SYSTEM CappingStation2
  (* Version 1.0, YYYY-MM-DD, Author, Eclipse 4diac *)
  APPLICATION Application
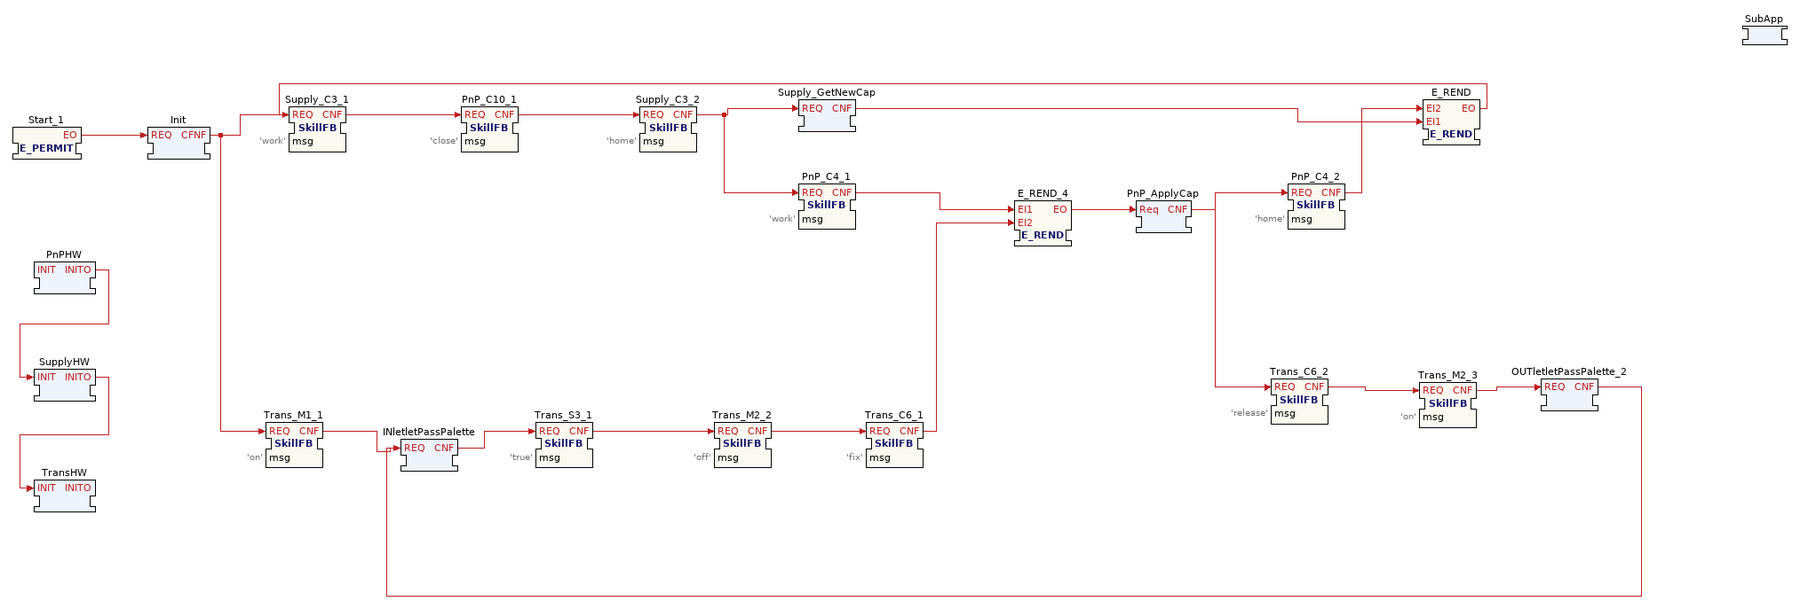
    FBS
      Start_1 : E_PERMIT;
      Supply_C3_1 : SkillFB(msg := 'work');
      Supply_C3_2 : SkillFB(msg := 'home');
      PnP_C10_1 : SkillFB(msg := 'close');
      PnP_C4_1 : SkillFB(msg := 'work');
      Trans_S3_1 : SkillFB(msg := 'true');
      Trans_M1_1 : SkillFB(msg := 'on');
      Trans_M2_2 : SkillFB(msg := 'off');
      Trans_C6_1 : SkillFB(msg := 'fix');
      E_REND_4 : E_REND;
      Trans_C6_2 : SkillFB(msg := 'release');
      Trans_M2_3 : SkillFB(msg := 'on');
      PnP_C4_2 : SkillFB(msg := 'home');
      E_REND : E_REND;
    END_FBS
    SUBAPPLICATION PnPHW
      EVENT_INPUT
        INIT;
      END_EVENT
      EVENT_OUTPUT
        INITO;
      END_EVENT
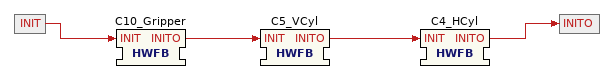
      FBS
        C10_Gripper : HWFB;
        C5_VCyl : HWFB;
        C4_HCyl : HWFB;
      END_FBS
      EVENT_CONNECTIONS
        INIT TO C10_Gripper.INIT;
        C10_Gripper.INITO TO C5_VCyl.INIT;
        C5_VCyl.INITO TO C4_HCyl.INIT;
        C4_HCyl.INITO TO INITO;
      END_CONNECTIONS
    END_SUBAPPLICATION
    SUBAPPLICATION SupplyHW
      EVENT_INPUT
        INIT;
      END_EVENT
      EVENT_OUTPUT
        INITO;
      END_EVENT
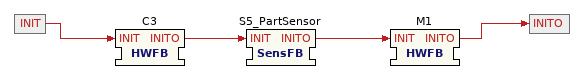
      FBS
        C3 : HWFB;
        M1 : HWFB;
        S5_PartSensor : SensFB;
      END_FBS
      EVENT_CONNECTIONS
        INIT TO C3.INIT;
        M1.INITO TO INITO;
        C3.INITO TO S5_PartSensor.INIT;
        S5_PartSensor.INITO TO M1.INIT;
      END_CONNECTIONS
    END_SUBAPPLICATION
    SUBAPPLICATION TransHW
      EVENT_INPUT
        INIT;
      END_EVENT
      EVENT_OUTPUT
        INITO;
      END_EVENT
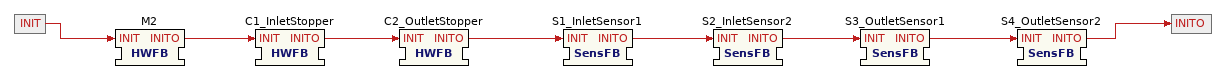
      FBS
        M2 : HWFB;
        C2_OutletStopper : HWFB;
        C1_InletStopper : HWFB;
        S1_InletSensor1 : SensFB;
        S2_InletSensor2 : SensFB;
        S3_OutletSensor1 : SensFB;
        S4_OutletSensor2 : SensFB;
      END_FBS
      EVENT_CONNECTIONS
        INIT TO M2.INIT;
        C1_InletStopper.INITO TO C2_OutletStopper.INIT;
        M2.INITO TO C1_InletStopper.INIT;
        C2_OutletStopper.INITO TO S1_InletSensor1.INIT;
        S1_InletSensor1.INITO TO S2_InletSensor2.INIT;
        S2_InletSensor2.INITO TO S3_OutletSensor1.INIT;
        S3_OutletSensor1.INITO TO S4_OutletSensor2.INIT;
        S4_OutletSensor2.INITO TO INITO;
      END_CONNECTIONS
    END_SUBAPPLICATION
    SUBAPPLICATION SubApp (* All Basic Skills *)
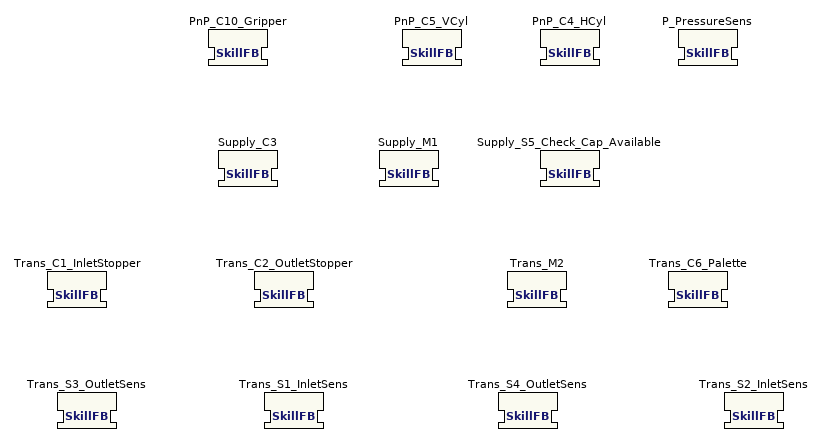
      FBS
        PnP_C10_Gripper : SkillFB;
        PnP_C5_VCyl : SkillFB;
        PnP_C4_HCyl : SkillFB;
        P_PressureSens : SkillFB;
        Supply_C3 : SkillFB;
        Supply_M1 : SkillFB;
        Supply_S5_Check_Cap_Available : SkillFB;
        Trans_C1_InletStopper : SkillFB;
        Trans_C2_OutletStopper : SkillFB;
        Trans_M2 : SkillFB;
        Trans_C6_Palette : SkillFB;
        Trans_S3_OutletSens : SkillFB;
        Trans_S4_OutletSens : SkillFB;
        Trans_S2_InletSens : SkillFB;
        Trans_S1_InletSens : SkillFB;
      END_FBS
    END_SUBAPPLICATION
    SUBAPPLICATION INletletPassPalette (* Composite Skill to let a product pass through the stoper *)
      EVENT_INPUT
        REQ;
      END_EVENT
      EVENT_OUTPUT
        CNF;
      END_EVENT
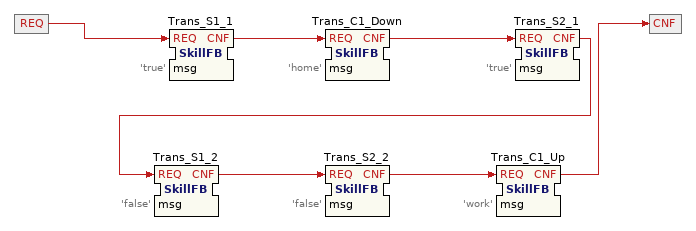
      FBS
        Trans_S1_2 : SkillFB(msg := 'false');
        Trans_S2_2 : SkillFB(msg := 'false');
        Trans_S1_1 : SkillFB(msg := 'true');
        Trans_S2_1 : SkillFB(msg := 'true');
        Trans_C1_Down : SkillFB(msg := 'home');
        Trans_C1_Up : SkillFB(msg := 'work');
      END_FBS
      EVENT_CONNECTIONS
        Trans_S1_2.CNF TO Trans_S2_2.REQ;
        Trans_S1_1.CNF TO Trans_C1_Down.REQ;
        Trans_C1_Down.CNF TO Trans_S2_1.REQ;
        REQ TO Trans_S1_1.REQ;
        Trans_S2_2.CNF TO Trans_C1_Up.REQ;
        Trans_C1_Up.CNF TO CNF;
        Trans_S2_1.CNF TO Trans_S1_2.REQ;
      END_CONNECTIONS
    END_SUBAPPLICATION
    SUBAPPLICATION OUTletletPassPalette_2
      EVENT_INPUT
        REQ;
      END_EVENT
      EVENT_OUTPUT
        CNF;
      END_EVENT
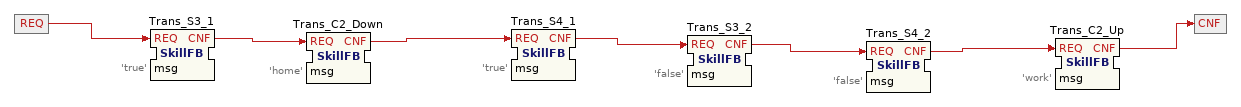
      FBS
        Trans_S3_2 : SkillFB(msg := 'false');
        Trans_S4_2 : SkillFB(msg := 'false');
        Trans_S3_1 : SkillFB(msg := 'true');
        Trans_S4_1 : SkillFB(msg := 'true');
        Trans_C2_Down : SkillFB(msg := 'home');
        Trans_C2_Up : SkillFB(msg := 'work');
      END_FBS
      EVENT_CONNECTIONS
        Trans_S4_1.CNF TO Trans_S3_2.REQ;
        Trans_S3_2.CNF TO Trans_S4_2.REQ;
        Trans_S3_1.CNF TO Trans_C2_Down.REQ;
        Trans_C2_Down.CNF TO Trans_S4_1.REQ;
        REQ TO Trans_S3_1.REQ;
        Trans_S4_2.CNF TO Trans_C2_Up.REQ;
        Trans_C2_Up.CNF TO CNF;
      END_CONNECTIONS
    END_SUBAPPLICATION
    SUBAPPLICATION Init
      EVENT_INPUT
        REQ;
      END_EVENT
      EVENT_OUTPUT
        CFNF;
      END_EVENT
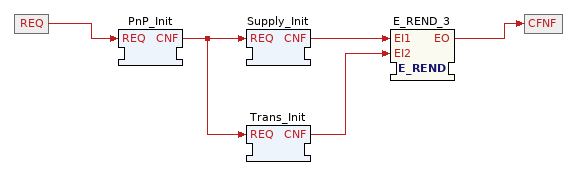
      FBS
        E_REND_3 : E_REND;
      END_FBS
      SUBAPPLICATION Supply_Init
        EVENT_INPUT
          REQ;
        END_EVENT
        EVENT_OUTPUT
          CNF;
        END_EVENT
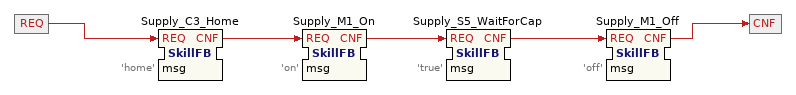
        FBS
          Supply_C3_Home : SkillFB(msg := 'home');
          Supply_M1_Off : SkillFB(msg := 'off');
          Supply_M1_On : SkillFB(msg := 'on');
          Supply_S5_WaitForCap : SkillFB(msg := 'true');
        END_FBS
        EVENT_CONNECTIONS
          Supply_C3_Home.CNF TO Supply_M1_On.REQ;
          Supply_S5_WaitForCap.CNF TO Supply_M1_Off.REQ;
          Supply_M1_On.CNF TO Supply_S5_WaitForCap.REQ;
          REQ TO Supply_C3_Home.REQ;
          Supply_M1_Off.CNF TO CNF;
        END_CONNECTIONS
      END_SUBAPPLICATION
      SUBAPPLICATION PnP_Init
        EVENT_INPUT
          REQ;
        END_EVENT
        EVENT_OUTPUT
          CNF;
        END_EVENT
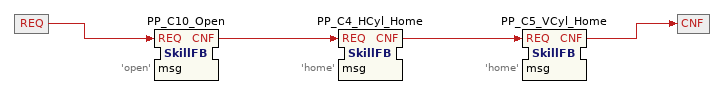
        FBS
          PP_C5_VCyl_Home : SkillFB(msg := 'home');
          PP_C4_HCyl_Home : SkillFB(msg := 'home');
          PP_C10_Open : SkillFB(msg := 'open');
        END_FBS
        EVENT_CONNECTIONS
          PP_C4_HCyl_Home.CNF TO PP_C5_VCyl_Home.REQ;
          PP_C10_Open.CNF TO PP_C4_HCyl_Home.REQ;
          PP_C5_VCyl_Home.CNF TO CNF;
          REQ TO PP_C10_Open.REQ;
        END_CONNECTIONS
      END_SUBAPPLICATION
      SUBAPPLICATION Trans_Init
        EVENT_INPUT
          REQ;
        END_EVENT
        EVENT_OUTPUT
          CNF;
        END_EVENT
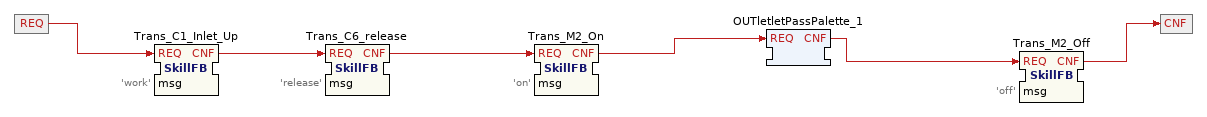
        FBS
          Trans_C1_Inlet_Up : SkillFB(msg := 'work');
          Trans_M2_On : SkillFB(msg := 'on');
          Trans_C6_release : SkillFB(msg := 'release');
          Trans_M2_Off : SkillFB(msg := 'off');
        END_FBS
        SUBAPPLICATION OUTletletPassPalette_1
          EVENT_INPUT
            REQ;
          END_EVENT
          EVENT_OUTPUT
            CNF;
          END_EVENT
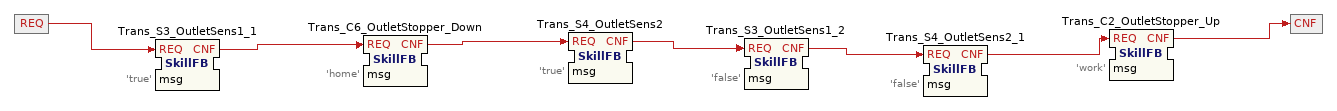
          FBS
            Trans_S3_OutletSens1_2 : SkillFB(msg := 'false');
            Trans_S4_OutletSens2_1 : SkillFB(msg := 'false');
            Trans_S3_OutletSens1_1 : SkillFB(msg := 'true');
            Trans_S4_OutletSens2 : SkillFB(msg := 'true');
            Trans_C6_OutletStopper_Down : SkillFB(msg := 'home');
            Trans_C2_OutletStopper_Up : SkillFB(msg := 'work');
          END_FBS
          EVENT_CONNECTIONS
            Trans_S4_OutletSens2.CNF TO Trans_S3_OutletSens1_2.REQ;
            Trans_S3_OutletSens1_2.CNF TO Trans_S4_OutletSens2_1.REQ;
            Trans_S3_OutletSens1_1.CNF TO Trans_C6_OutletStopper_Down.REQ;
            Trans_C6_OutletStopper_Down.CNF TO Trans_S4_OutletSens2.REQ;
            REQ TO Trans_S3_OutletSens1_1.REQ;
            Trans_S4_OutletSens2_1.CNF TO Trans_C2_OutletStopper_Up.REQ;
            Trans_C2_OutletStopper_Up.CNF TO CNF;
          END_CONNECTIONS
        END_SUBAPPLICATION
        EVENT_CONNECTIONS
          Trans_C1_Inlet_Up.CNF TO Trans_C6_release.REQ;
          Trans_C6_release.CNF TO Trans_M2_On.REQ;
          REQ TO Trans_C1_Inlet_Up.REQ;
          Trans_M2_On.CNF TO OUTletletPassPalette_1.REQ;
          Trans_M2_Off.CNF TO CNF;
          OUTletletPassPalette_1.CNF TO Trans_M2_Off.REQ;
        END_CONNECTIONS
      END_SUBAPPLICATION
      EVENT_CONNECTIONS
        PnP_Init.CNF TO Supply_Init.REQ;
        Supply_Init.CNF TO E_REND_3.EI1;
        PnP_Init.CNF TO Trans_Init.REQ;
        Trans_Init.CNF TO E_REND_3.EI2;
        REQ TO PnP_Init.REQ;
        E_REND_3.EO TO CFNF;
      END_CONNECTIONS
    END_SUBAPPLICATION
    SUBAPPLICATION PnP_ApplyCap
      EVENT_INPUT
        Req;
      END_EVENT
      EVENT_OUTPUT
        CNF;
      END_EVENT
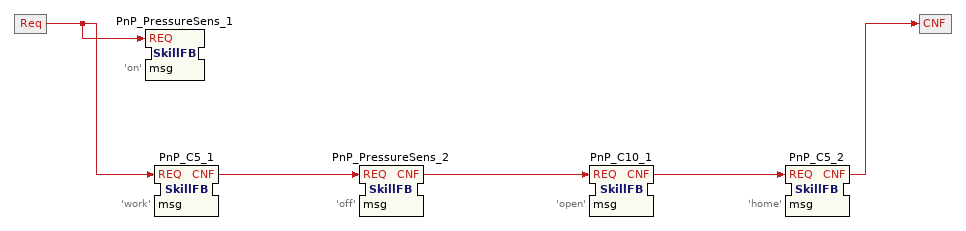
      FBS
        PnP_PressureSens_1 : SkillFB(msg := 'on');
        PnP_C10_1 : SkillFB(msg := 'open');
        PnP_PressureSens_2 : SkillFB(msg := 'off');
        PnP_C5_2 : SkillFB(msg := 'home');
        PnP_C5_1 : SkillFB(msg := 'work');
      END_FBS
      EVENT_CONNECTIONS
        PnP_PressureSens_2.CNF TO PnP_C10_1.REQ;
        PnP_C10_1.CNF TO PnP_C5_2.REQ;
        PnP_C5_1.CNF TO PnP_PressureSens_2.REQ;
        Req TO PnP_PressureSens_1.REQ;
        PnP_C5_2.CNF TO CNF;
        Req TO PnP_C5_1.REQ;
      END_CONNECTIONS
    END_SUBAPPLICATION
    SUBAPPLICATION Supply_GetNewCap
      EVENT_INPUT
        REQ;
      END_EVENT
      EVENT_OUTPUT
        CNF;
      END_EVENT
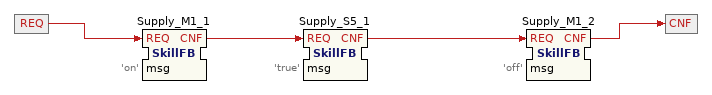
      FBS
        Supply_M1_2 : SkillFB(msg := 'off');
        Supply_M1_1 : SkillFB(msg := 'on');
        Supply_S5_1 : SkillFB(msg := 'true');
      END_FBS
      EVENT_CONNECTIONS
        Supply_S5_1.CNF TO Supply_M1_2.REQ;
        Supply_M1_1.CNF TO Supply_S5_1.REQ;
        Supply_M1_2.CNF TO CNF;
        REQ TO Supply_M1_1.REQ;
      END_CONNECTIONS
    END_SUBAPPLICATION
    EVENT_CONNECTIONS
      PnPHW.INITO TO SupplyHW.INIT;
      Supply_C3_1.CNF TO PnP_C10_1.REQ;
      PnP_C10_1.CNF TO Supply_C3_2.REQ;
      Supply_C3_2.CNF TO PnP_C4_1.REQ;
      INletletPassPalette.CNF TO Trans_S3_1.REQ;
      Trans_S3_1.CNF TO Trans_M2_2.REQ;
      Trans_M2_2.CNF TO Trans_C6_1.REQ;
      PnP_C4_1.CNF TO E_REND_4.EI1;
      Trans_C6_1.CNF TO E_REND_4.EI2;
      Trans_C6_2.CNF TO Trans_M2_3.REQ;
      Trans_M2_3.CNF TO OUTletletPassPalette_2.REQ;
      OUTletletPassPalette_2.CNF TO INletletPassPalette.REQ;
      PnP_C4_2.CNF TO E_REND.EI2;
      Start_1.EO TO Init.REQ;
      Init.CFNF TO Supply_C3_1.REQ;
      Init.CFNF TO Trans_M1_1.REQ;
      E_REND.EO TO Supply_C3_1.REQ;
      Trans_M1_1.CNF TO INletletPassPalette.REQ;
      PnP_ApplyCap.CNF TO Trans_C6_2.REQ;
      PnP_ApplyCap.CNF TO PnP_C4_2.REQ;
      Supply_GetNewCap.CNF TO E_REND.EI1;
      Supply_C3_2.CNF TO Supply_GetNewCap.REQ;
      E_REND_4.EO TO PnP_ApplyCap.Req;
      SupplyHW.INITO TO TransHW.INIT;
    END_CONNECTIONS
  END_APPLICATION
  DEVICE PnP_Unit : FORTE_PC(MGR_ID := "localhost:61499")
    {SET_ATTRIBUTE(Profile, HOLOBLOC)} (* device profile *)
    RESOURCE EMB_RES : EMB_RES
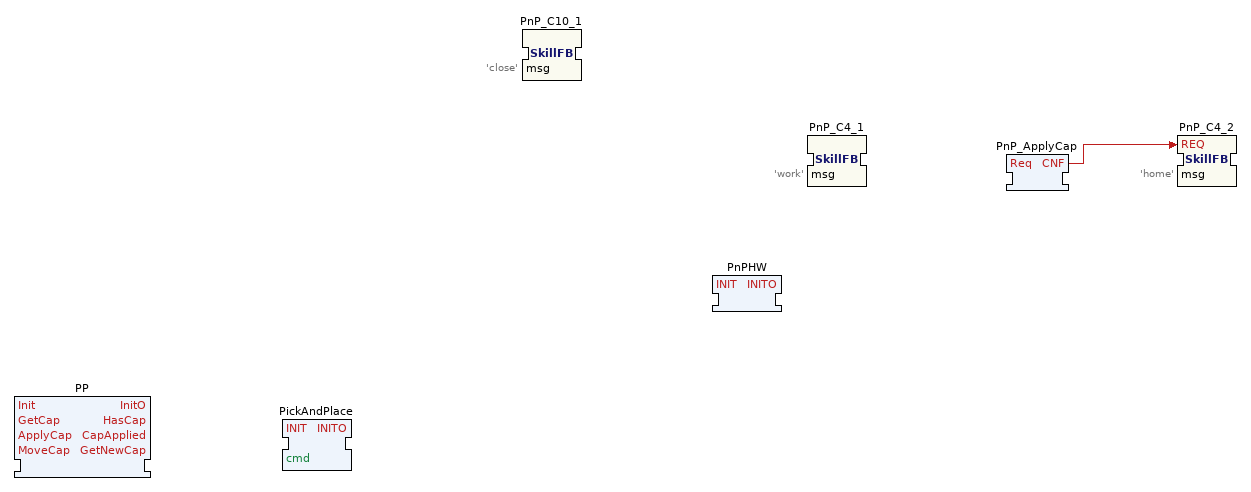
      FBS
        PnP_C10_1 : SkillFB(msg := 'close');
        PnP_C4_1 : SkillFB(msg := 'work');
        PnP_C4_2 : SkillFB(msg := 'home');
      END_FBS
      SUBAPPLICATION PnPHW
        EVENT_INPUT
          INIT;
        END_EVENT
        EVENT_OUTPUT
          INITO;
        END_EVENT
      END_SUBAPPLICATION
      SUBAPPLICATION PnP_ApplyCap
        EVENT_INPUT
          Req;
        END_EVENT
        EVENT_OUTPUT
          CNF;
        END_EVENT
      END_SUBAPPLICATION
      SUBAPPLICATION PP
        EVENT_INPUT
          Init;
          GetCap;
          ApplyCap;
          MoveCap;
        END_EVENT
        EVENT_OUTPUT
          InitO;
          HasCap;
          CapApplied;
          GetNewCap;
        END_EVENT
      END_SUBAPPLICATION
      SUBAPPLICATION PickAndPlace
        EVENT_INPUT
          INIT;
        END_EVENT
        EVENT_OUTPUT
          INITO;
        END_EVENT
        SOCKETS
          cmd : APickNPlace;
        END_SOCKETS
      END_SUBAPPLICATION
      EVENT_CONNECTIONS
        PnP_ApplyCap.CNF TO PnP_C4_2.REQ;
      END_CONNECTIONS
    END_RESOURCE
  END_DEVICE
  DEVICE Supply_Unit : FORTE_PC(MGR_ID := "localhost:61499")
    {SET_ATTRIBUTE(Profile, HOLOBLOC)} (* device profile *)
    RESOURCE EMB_RES : EMB_RES
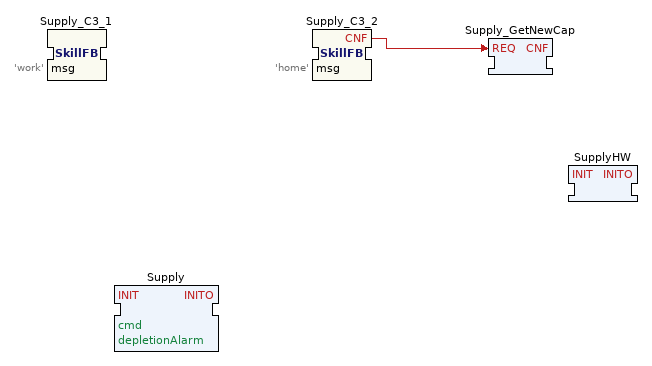
      FBS
        Supply_C3_1 : SkillFB(msg := 'work');
        Supply_C3_2 : SkillFB(msg := 'home');
      END_FBS
      SUBAPPLICATION Supply
        EVENT_INPUT
          Init;
          ProvideCap;
          PPTookCap;
        END_EVENT
        EVENT_OUTPUT
          InitO;
          CapAvailable;
          PPCanMove;
        END_EVENT
      END_SUBAPPLICATION
      SUBAPPLICATION Supply
        EVENT_INPUT
          INIT;
        END_EVENT
        EVENT_OUTPUT
          INITO;
        END_EVENT
        SOCKETS
          cmd : ASupply;
          depletionAlarm : Alarm;
        END_SOCKETS
      END_SUBAPPLICATION
      SUBAPPLICATION Supply_GetNewCap
        EVENT_INPUT
          REQ;
        END_EVENT
        EVENT_OUTPUT
          CNF;
        END_EVENT
      END_SUBAPPLICATION
      SUBAPPLICATION SupplyHW
        EVENT_INPUT
          INIT;
        END_EVENT
        EVENT_OUTPUT
          INITO;
        END_EVENT
      END_SUBAPPLICATION
      EVENT_CONNECTIONS
        Supply_C3_2.CNF TO Supply_GetNewCap.REQ;
      END_CONNECTIONS
    END_RESOURCE
  END_DEVICE
  DEVICE Transport_Unit : FORTE_PC(MGR_ID := "localhost:61499")
    {SET_ATTRIBUTE(Profile, HOLOBLOC)} (* device profile *)
    RESOURCE EMB_RES : EMB_RES
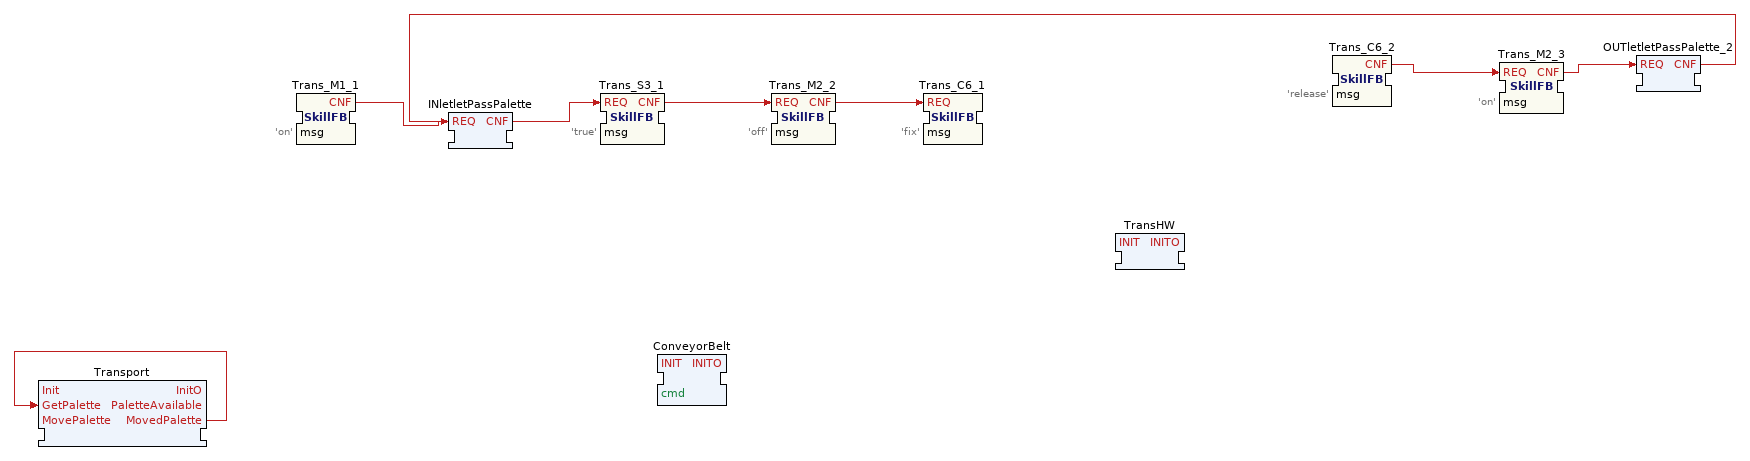
      FBS
        Trans_M2_3 : SkillFB(msg := 'on');
        Trans_C6_2 : SkillFB(msg := 'release');
        Trans_C6_1 : SkillFB(msg := 'fix');
        Trans_M2_2 : SkillFB(msg := 'off');
        Trans_S3_1 : SkillFB(msg := 'true');
        Trans_M1_1 : SkillFB(msg := 'on');
      END_FBS
      SUBAPPLICATION TransHW
        EVENT_INPUT
          INIT;
        END_EVENT
        EVENT_OUTPUT
          INITO;
        END_EVENT
      END_SUBAPPLICATION
      SUBAPPLICATION OUTletletPassPalette_2
        EVENT_INPUT
          REQ;
        END_EVENT
        EVENT_OUTPUT
          CNF;
        END_EVENT
      END_SUBAPPLICATION
      SUBAPPLICATION INletletPassPalette
        EVENT_INPUT
          REQ;
        END_EVENT
        EVENT_OUTPUT
          CNF;
        END_EVENT
      END_SUBAPPLICATION
      SUBAPPLICATION Transport
        EVENT_INPUT
          Init;
          GetPalette;
          MovePalette;
        END_EVENT
        EVENT_OUTPUT
          InitO;
          PaletteAvailable;
          MovedPalette;
        END_EVENT
      END_SUBAPPLICATION
      SUBAPPLICATION ConveyorBelt
        EVENT_INPUT
          INIT;
        END_EVENT
        EVENT_OUTPUT
          INITO;
        END_EVENT
        SOCKETS
          cmd : AConveyor;
        END_SOCKETS
      END_SUBAPPLICATION
      EVENT_CONNECTIONS
        Trans_M2_3.CNF TO OUTletletPassPalette_2.REQ;
        Trans_C6_2.CNF TO Trans_M2_3.REQ;
        Trans_M2_2.CNF TO Trans_C6_1.REQ;
        Trans_S3_1.CNF TO Trans_M2_2.REQ;
        OUTletletPassPalette_2.CNF TO INletletPassPalette.REQ;
        Trans_M1_1.CNF TO INletletPassPalette.REQ;
        INletletPassPalette.CNF TO Trans_S3_1.REQ;
        Transport.MovedPalette TO Transport.GetPalette;
      END_CONNECTIONS
    END_RESOURCE
  END_DEVICE
  MAPPINGS
    Application.Supply_C3_1 ON Supply_Unit.EMB_RES.Supply_C3_1;
    Application.Supply_C3_2 ON Supply_Unit.EMB_RES.Supply_C3_2;
    Application.PnPHW ON PnP_Unit.EMB_RES.PnPHW;
    Application.PnP_C10_1 ON PnP_Unit.EMB_RES.PnP_C10_1;
    Application.PnP_C4_1 ON PnP_Unit.EMB_RES.PnP_C4_1;
    Application.PnP_ApplyCap ON PnP_Unit.EMB_RES.PnP_ApplyCap;
    Application.PnP_C4_2 ON PnP_Unit.EMB_RES.PnP_C4_2;
    Application.TransHW ON Transport_Unit.EMB_RES.TransHW;
    Application.OUTletletPassPalette_2 ON Transport_Unit.EMB_RES.OUTletletPassPalette_2;
    Application.Trans_M2_3 ON Transport_Unit.EMB_RES.Trans_M2_3;
    Application.Trans_C6_2 ON Transport_Unit.EMB_RES.Trans_C6_2;
    Application.Trans_C6_1 ON Transport_Unit.EMB_RES.Trans_C6_1;
    Application.Trans_M2_2 ON Transport_Unit.EMB_RES.Trans_M2_2;
    Application.Trans_S3_1 ON Transport_Unit.EMB_RES.Trans_S3_1;
    Application.Trans_M1_1 ON Transport_Unit.EMB_RES.Trans_M1_1;
    Application.INletletPassPalette ON Transport_Unit.EMB_RES.INletletPassPalette;
    Application.Supply_GetNewCap ON Supply_Unit.EMB_RES.Supply_GetNewCap;
    Application.SupplyHW ON Supply_Unit.EMB_RES.SupplyHW;
  END_MAPPINGS
  SEGMENTS
    Ethernet : Ethernet;
  END_SEGMENTS
  LINKS
    Supply_Unit => Ethernet;
    PnP_Unit => Ethernet;
    Transport_Unit => Ethernet;
  END_LINKS
END_SYSTEM
